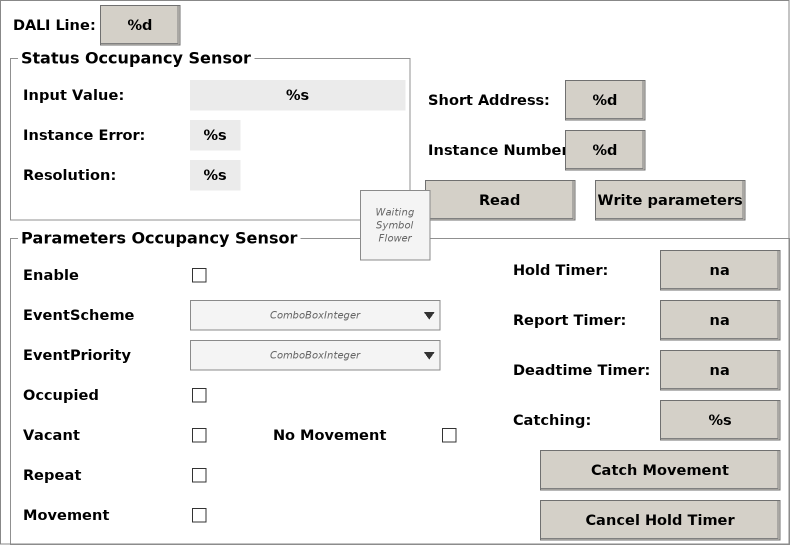
VISUALIZATION Visu_Part303OccupancySensor  // 790x545
    GroupBox (10,230 780x315), "Parameters Occupancy Sensor"
        Button (650,70 120x40), "%d s", text variable: DALI_Commissioning.fbPart303OccupancySensor.nReport
            OnMouseClick: write the text variable via Default, min 0, max 255, title "Insert value for report timer"
        Button (650,70 120x40), "na", invisible if: Not DALI_Commissioning.fbPart303OccupancySensor.bNoReportTimer, input disabled if: Not DALI_Commissioning.fbPart303OccupancySensor.bNoReportTimer
        Textfield (500,125 145x30), "Deadtime Timer:"
        Textfield (500,75 145x30), "Report Timer:"
        Textfield (500,25 145x30), "Hold Timer:"
        Button (650,20 120x40), "%d s", text variable: DALI_Commissioning.fbPart303OccupancySensor.nHold, invisible if: DALI_Commissioning.fbPart303OccupancySensor.bNoHoldTimer, input disabled if: DALI_Commissioning.fbPart303OccupancySensor.bNoHoldTimer
            OnMouseClick: write the text variable via Default, min 0, max 2538, title "Insert value for hold timer"
        Textfield (10,30 150x30), "Enable"
        Button (650,120 120x40), "%d ms", text variable: DALI_Commissioning.fbPart303OccupancySensor.nDeadtime
            OnMouseClick: write the text variable via Default, min 0, max 12750, title "Insert value for deadtime timer"
        Checkbox (180,30 30x30), variable: DALI_Commissioning.fbPart303OccupancySensor.bEnable
        Textfield (10,70 150x30), "EventScheme"
        Textfield (10,150 150x30), "Occupied"
        Textfield (10,190 150x30), "Vacant"
        Textfield (10,230 150x30), "Repeat"
        Textfield (10,270 150x30), "Movement"
        Textfield (260,190 150x30), "No Movement"
        Checkbox (180,150 30x30), variable: DALI_Commissioning.fbPart303OccupancySensor.bOccupied
        Checkbox (180,190 30x30), variable: DALI_Commissioning.fbPart303OccupancySensor.bVacant
        Checkbox (180,230 30x30), variable: DALI_Commissioning.fbPart303OccupancySensor.bRepeat
        Checkbox (430,190 30x30), variable: DALI_Commissioning.fbPart303OccupancySensor.bNoMovement
        ComboBoxInteger (180,70 250x30), variable: DALI_Commissioning.fbPart303OccupancySensor.eEventScheme, text list: 'EventScheme'
        Checkbox (180,270 30x30), variable: DALI_Commissioning.fbPart303OccupancySensor.bMovement
        Button (650,120 120x40), "na", invisible if: Not DALI_Commissioning.fbPart303OccupancySensor.bNoDeadtimeTimer, input disabled if: Not DALI_Commissioning.fbPart303OccupancySensor.bNoDeadtimeTimer
        Button (530,270 240x40), "Cancel Hold Timer"
            OnMouseClick: execute { DALI_Commissioning.fbPart303OccupancySensor.bCancelHoldTimer := true; }
        Textfield (10,110 150x30), "EventPriority"
        ComboBoxInteger (180,110 250x30), variable: DALI_Commissioning.fbPart303OccupancySensor.eEventPriority, text list: 'EventPriority'
        Button (650,20 120x40), "na", invisible if: Not DALI_Commissioning.fbPart303OccupancySensor.bNoHoldTimer, input disabled if: Not DALI_Commissioning.fbPart303OccupancySensor.bNoHoldTimer
        Button (530,220 240x40), "Catch Movement"
            OnMouseClick: execute { DALI_Commissioning.fbPart303OccupancySensor.bCatchMovement := true; }
        Textfield (500,175 145x30), "Catching:"
    GroupBox (10,50 400x170), "Status Occupancy Sensor"
        Textfield (10,30 160x30), "Input Value:"
        Textfield (10,70 160x30), "Instance Error:"
        Textfield (10,110 160x30), "Resolution:"
        Textfield (180,30 215x30), "%s", text variable: DALI_Commissioning.fbPart303OccupancySensor.sInputValue
        Textfield (180,70 50x30), "%s", text variable: DALI_Commissioning.fbPart303OccupancySensor.nInstanceError
        Textfield (180,110 50x30), "%s", text variable: DALI_Commissioning.fbPart303OccupancySensor.nResolution
    Button (425,180 150x40), "Read"
        OnMouseClick: execute { DALI_Commissioning.fbPart303OccupancySensor.bRead := TRUE; }
    WaitingSymbolFlower (360,190 70x70), invisible if: DALI_Commissioning.fbPart303OccupancySensor.bHideWaitSymbol
    Button (595,180 150x40), "Write parameters"
        OnMouseClick: execute { DALI_Commissioning.fbPart303OccupancySensor.bWrite := TRUE; }
    Button (660,400 120x40), "%s", text variable: DALI_Commissioning.fbPart303OccupancySensor.sCatching
        OnMouseClick: write the text variable via Default, min 0, max 12750, title "Insert value for deadtime timer"
    Group (10,5 170x40)
        Textfield (0,0 110x40), "DALI Line:"
        Button (90,0 80x40), "%d", text variable: GVL_Internal.nDALILine
            OnMouseClick: write the text variable via Default, min 1, max 10, title "Choose line"
    Textfield (425,80 130x40), "Short Address:"
    Button (565,80 80x40), "%d", text variable: DALI_Commissioning.fbPart303OccupancySensor.nAddress
        OnMouseClick: write the text variable via Default, min 0, max 63, title "Insert Short Address"
    Textfield (425,130 150x40), "Instance Number:"
    Button (565,130 80x40), "%d", text variable: DALI_Commissioning.fbPart303OccupancySensor.nInstanceAddress
        OnMouseClick: write the text variable via Default, min 0, max 31, title "Insert instance number"
END_VISUALIZATION

(* stored: Version 1.1.0.1
   Visu Visu_Part303OccupancySensor: Id {fe3851b5-d5a0-4e49-8a23-d370abf5a4bc} *)
